# EPICS substitutions: streamApp/pluginDb/commonPlugins.substitutions
# commonPlugins.substitutions
# TODO: Combine all the substitution files for the plugins in commonPlugins.cmd
# here to create one commonPlugins.db
#

file cross.template
{
    pattern
    {   N,  P,          R   }
    {   1,  "$(CAM):",  ""  }
    {   2,  "$(CAM):",  ""  }
    {   3,  "$(CAM):",  ""  }
    {   4,  "$(CAM):",  ""  }
}
